DATA_BLOCK "dbArchiveEquipRectifier"
{ S7_Optimized_Access := 'TRUE' }
VERSION : 0.8
NON_RETAIN
"fbArchiveEquipRectifier"

BEGIN

END_DATA_BLOCK

